FUNCTION_BLOCK FB_SaMElementHolding EXTENDS FB_SaMElement
VAR
END_VAR

METHOD FB_init : BOOL
VAR_INPUT
	bInitRetains : BOOL; // if TRUE, the retain variables are initialized (warm start / cold start)
	bInCopyCode : BOOL;  // if TRUE, the instance afterwards gets moved into the copy code (online change)
END_VAR
THIS^.SetText (eLocation := E_BaseLocation.pl, wsDescription := "Wstrzymywanie");
THIS^.SetText (eLocation := E_BaseLocation.en, wsDescription := "Holding");
THIS^.SetText (eLocation := E_BaseLocation.de, wsDescription := "Halten");
THIS^.SetName (stName := THIS^.GetTexts ());
END_METHOD

METHOD PUBLIC InvokeStateForTopElement : BOOL
VAR_INPUT
	itfTopElement		: ITF_BaseSaMStateMethod;
END_VAR
InvokeStateForTopElement	:= itfTopElement.SP_Holding ();
END_METHOD

END_FUNCTION_BLOCK

(* stored: Version 1.1.0.1
   POU FB_SaMElementHolding: Id {5dbc55bf-d793-0fb3-399d-491cc4b2743a}, SpecialFunc None
   Method FB_init: Id {d14c10d4-e703-0002-35a6-5f25e9ae0e7e}
   Method InvokeStateForTopElement: Id {d9fdbde0-928d-09ae-0609-b6b9dcb878fb} *)
